// TwinCAT 3 PLC project Structures
// ProgramVersion: 3.1.4023.0
// libraries:
//   Tc2_Standard, * (Beckhoff Automation GmbH)
//   Tc2_System, * (Beckhoff Automation GmbH)
//   Tc3_Module, * (Beckhoff Automation GmbH)
// project tree:
//   DUTs/ ST_Event.TcDUT
//   / PlcTask.TcTTO
//   POUs/ MAIN.TcPOU, UpdateEventTimestampWithSystemTime.TcPOU
// (motion and I/O tree: see PLC project arrays1)
// real-time tasks:
//   TASK PlcTask: cycle T#10ms, priority 20, ADS port 350
//   TASK PlcTask1: cycle T#10ms, priority 21, ADS port 351
//   TASK PlcTask2: cycle T#10ms, priority 22, ADS port 352
//   TASK PlcTask3: cycle T#10ms, priority 23, ADS port 353

CONFIGURATION Structures
    RESOURCE PLC ON TwinCAT3
        TASK PlcTask(INTERVAL := T#10ms, PRIORITY := 21);
        PROGRAM MAIN WITH PlcTask : MAIN;
    END_RESOURCE
END_CONFIGURATION

// ---- DUTs/ST_Event.TcDUT
TYPE ST_Event :
STRUCT
	eEventType : E_EventType;
	eEventSeverity : TcEventSeverity;
	nEventIdentity : UDINT;
	sEventText : STRING(255);
	dtTimestamp : DATE_AND_TIME;
END_STRUCT
END_TYPE

// ---- POUs/MAIN.TcPOU
PROGRAM MAIN
VAR
	aEvents : ARRAY[1..100] OF ST_Event;
	sTempString : STRING(255);
END_VAR

sTempString := aEvents[33].sEventText;

END_PROGRAM

// ---- POUs/UpdateEventTimestampWithSystemTime.TcPOU
FUNCTION UpdateEventTimestampWithSystemTime
VAR_INPUT
	stEvent : ST_Event;
END_VAR
VAR_OUTPUT
	stEventOut : ST_Event;
END_VAR

(*Pass by value*)
stEventOut := stEvent;
stEventOut.dtTimestamp := // ...(GetSystemTime...)

END_FUNCTION
